ABB RobotStudio station: task_1.rspag

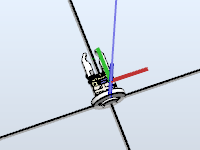
Station Station (saved by RobotStudio 7.0.8746.631)
Layout (positions relative to the parent item):
  - Gripper [mechanism] at (0, 0, 0) mm; joint values [0, 0] (rad or m)
      TCP tGripper at (0, 0, 72) mm
      links: L1, A, B
